(* IEC 61131-3 sources: UniTest/UniTest_br/Library_tests/test_assertGreater_UDINT, 1 file *)

(* ---- main.st ---- *)
PROGRAM _CYCLIC
    (*https://github.com/tkucic/UniTest/blob/main/docs/docs/ns/Library_tests/prg/test_assertGreater_UDINT.md*)
    (*Run the test cases*)
    TEST_CASE_1_SETUP;
    TEST_CASE_1_EXEC;

    TEST_CASE_2_SETUP;
    TEST_CASE_2_EXEC;

    (*Instantiate the test runner*)
    testRunner(
    	Id := 59,
    	Name := 'assertGreater_UDINT',
        RunTests := gRunAll OR vRunAll,
    	ResetTests := gResetAll OR vResetAll,
    	TestCases:=vTestCases);

    (*Report the results to the collection global*)
    gResults[testRunner.Id] := testRunner.Summary;
END_PROGRAM
